{attribute 'qualified_only'}
{attribute 'strict'}
{attribute 'to_string'}
TYPE cPuckSide :
(
	None := 0,
	Clean,
	Dirty
);
END_TYPE

(* stored: Version 1.1.0.1, ProductVersion 3.1.4024.6
   DUT cPuckSide: Id {6244c760-4710-4cbc-b178-40bc276ac41d} *)
